PROGRAM HouseControl
VAR

END_VAR


IF stTime.wHour = 18 AND stTime.wMinute =1 THEN
StairLight := TRUE; //Cant be shut off for 1 minute 
ELSIF stTime.wHour = 23 AND stTime.wMinute =59 THEN
StairLight := TRUE; //Cant be shut off for 1 minute 	
END_IF

END_PROGRAM

(* stored: Version 1.1.0.1, ProductVersion 3.1.4024.12
   POU HouseControl: Id {a1e03bf8-e102-41a7-ba3f-92cced89e329}, SpecialFunc None *)
